PROGRAM MAIN
VAR
	FirstAddedVariables : BOOL;
	SecondAdded : INT;
END_VAR

FirstAddedVariables := TRUE;

END_PROGRAM

(* stored: Version 1.1.0.1, ProductVersion 3.1.4024.6
   POU MAIN: Id {c3ec141f-da58-4d58-a482-7517298a7f1a}, SpecialFunc None *)
